Universal Robots PolyScope program: submain.urp

Program submain (installation=default directory=/programs/usbdisk_0 createdIn=5.13.0 lastSavedIn=5.13.0 robotSerialNumber=20195600261)
Calibrated DH parameters: a=[0.000314, -0.466486, -0.015685, 0.000033, 0.000024, 0]; d=[0.181135, -61.162157, 368.282682, -306.94627, 0.120009, 0.115625]; alpha=[1.570909, 0.001741, -0.001171, 1.570507, -1.571069, 0]; deltaTheta=[-0.000001, -0.224411, 4.980378, 1.52722, -0.000003, 0]
InitVariablesNode
BeforeStart
  jp_beck := rpc_factory("xmlrpc","http://10.2.4.106:33000")
Robot Program (runOnlyOnce=false)
  Wait Sleep waitTime=1
  Script: jp_beck.yuki_log(get_actual_tcp_pose(),"TCP")
